FUNCTION_BLOCK FB_InverBytesOrder_Test EXTENDS TcUnit.FB_TestSuite

TestWord('Invert WORD_1', nData := 16#1234, nExpected:= 16#3412);
TestWord('Invert WORD_2', nData := 16#4321, nExpected:= 16#2143);

TestDWord('Invert DWORD_1', nData := 16#12345678, nExpected:= 16#78563412);
TestDWord('Invert DWORD_2', nData := 16#87654321, nExpected:= 16#21436587);

TestLWord('Invert LWORD_1', nData := 16#1234567812345678, nExpected:= 16#7856341278563412);
TestLWord('Invert LWORD_2', nData := 16#8765432187654321, nExpected:= 16#2143658721436587);

METHOD TestDWord
VAR_INPUT
	sName : T_MaxString;	
	nData 	: DWORD;
	nExpected : DWORD;
END_VAR

VAR		
	nResult : DWORD;
END_VAR
TEST(sName);


F_InverBytesOrder(nData);
AssertEquals(Expected := nExpected,
             Actual := nData,
             Message := 'Result value is not correct');	
	 
TEST_FINISHED();
END_METHOD

METHOD TestLWord
VAR_INPUT
	sName : T_MaxString;	
	nData 	: LWORD;
	nExpected : LWORD;
END_VAR

VAR		
	nResult : LWORD;
END_VAR
TEST(sName);


F_InverBytesOrder(nData);
AssertEquals(Expected := nExpected,
             Actual := nData,
             Message := 'Result value is not correct');	
	 
TEST_FINISHED();
END_METHOD

METHOD TestWord
VAR_INPUT
	sName : T_MaxString;	
	nData 	: WORD;
	nExpected : WORD;
END_VAR

VAR		
	nResult : WORD;
END_VAR
TEST(sName);


F_InverBytesOrder(nData);
AssertEquals(Expected := nExpected,
             Actual := nData,
             Message := 'Result value is not correct');	
	 
TEST_FINISHED();
END_METHOD

END_FUNCTION_BLOCK

(* stored: Version 1.1.0.1, ProductVersion 3.1.4024.12
   POU FB_InverBytesOrder_Test: Id {140c23b6-c900-0392-3cfd-b22c9301fc15}, SpecialFunc None
   Method TestDWord: Id {b3014372-fae4-02ff-0242-ab66131b9271}
   Method TestLWord: Id {4460bd71-9918-088c-31e6-d81993e65c66}
   Method TestWord: Id {66c44461-15cc-0aaf-1902-8868fd540106} *)
